TYPE ST_CenterPosition :
STRUCT
  Input : ST_PositionXY;
  Diagnose : ST_PositionXY;
END_STRUCT
END_TYPE

(* stored: Version 1.1.0.1, ProductVersion 3.1.4024.12
   DUT ST_CenterPosition: Id {01af67df-38fc-40aa-8c0e-04f1c6e2a525} *)
